(* Visualisation AMAININTERFACE
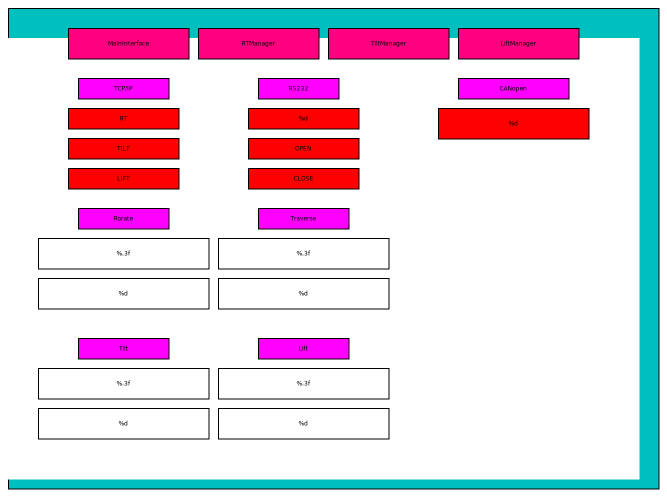
rounded rectangle at (60,20)-(181,51): text "MainInterface"; opens aMainInterface
rounded rectangle at (190,20)-(311,51): text "RTManager"; opens bRTManager
rounded rectangle at (320,20)-(441,51): text "TiltManager"; opens TiltManager
rounded rectangle at (450,20)-(571,51): text "LiftManager"; opens LiftManager
rounded rectangle at (450,70)-(561,91): text "CANopen"
rounded rectangle at (250,70)-(331,91): text "RS232"
rounded rectangle at (70,70)-(161,91): text "TCP/IP"
rounded rectangle at (70,200)-(161,221): text "Rorate"
rounded rectangle at (250,200)-(341,221): text "Traverse"
rounded rectangle at (70,330)-(161,351): text "Tilt"
rounded rectangle at (250,330)-(341,351): text "Lift"
rounded rectangle at (30,360)-(201,391): text "%.3f"
rounded rectangle at (210,360)-(381,391): text "%.3f"; shows .ENC_POS1/100.0
rounded rectangle at (30,400)-(201,431): text "%d"; shows .diActVelocity1/(-2000)
rounded rectangle at (210,400)-(381,431): text "%d"; shows .diActVelocity2/3360
rounded rectangle at (210,230)-(381,261): text "%.3f"; shows .ENC_POS1/100.0
rounded rectangle at (30,230)-(201,261): text "%.3f"
rounded rectangle at (30,270)-(201,301): text "%d"; shows .diActVelocity1/(-2000)
rounded rectangle at (210,270)-(381,301): text "%d"; shows .diActVelocity2/3360
rectangle at (430,100)-(581,131): text "%d"; shows pCanOpenNode[0].nStatus; alarm colour if pCanOpenNode[0].nStatus=5
rounded rectangle at (240,100)-(351,121): text "%d"; shows ComHandle; alarm colour if ComHandle>0
rounded rectangle at (240,130)-(351,151): text "OPEN"; alarm colour if PLC_PRG.open
rounded rectangle at (240,160)-(351,181): text "CLOSE"; alarm colour if PLC_PRG.close
rounded rectangle at (60,100)-(171,121): text "RT"; alarm colour if Client0.diSocket<>-1
rounded rectangle at (60,130)-(171,151): text "TILT"; alarm colour if Client1.diSocket<>-1
rounded rectangle at (60,160)-(171,181): text "LIFT"; alarm colour if Client2.diSocket<>-1
7 more shapes without text or variables
*)

(* Visualisation bRTManager
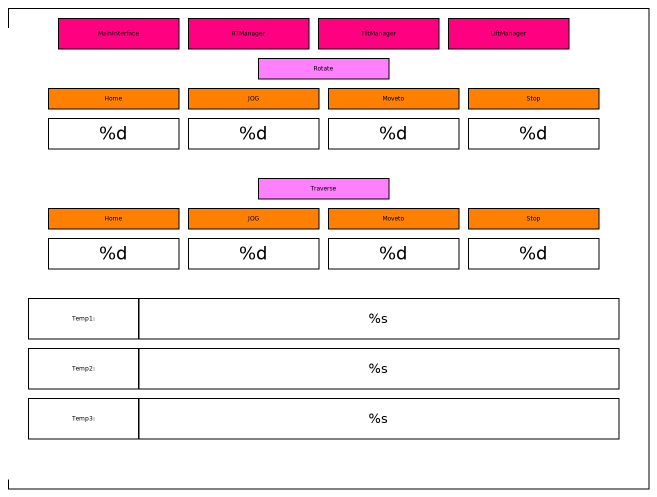
rectangle at (130,340)-(611,381): text "%s"; shows RT_Manager.Temp2
rectangle at (130,390)-(611,431): text "%s"; shows RT_Manager.Temp3
rectangle at (130,290)-(611,331): text "%s"; shows RT_Manager.Temp
rounded rectangle at (250,170)-(381,191): text "Traverse"
rounded rectangle at (40,200)-(171,221): text "Home"
rounded rectangle at (180,200)-(311,221): text "JOG"
rounded rectangle at (320,200)-(451,221): text "Moveto"
rounded rectangle at (460,200)-(591,221): text "Stop"
rectangle at (40,230)-(171,261): text "%d"; shows RT_Manager.diTraverseHomestep
rectangle at (180,230)-(311,261): text "%d"; shows RT_Manager.diTraverseJogstep
rectangle at (320,230)-(451,261): text "%d"; shows RT_Manager.diTraverseMovetostep
rectangle at (460,230)-(591,261): text "%d"; shows RT_Manager.diTraverseStopstep
rectangle at (20,290)-(131,331): text "Temp1:"
rectangle at (20,340)-(131,381): text "Temp2:"
rectangle at (20,390)-(131,431): text "Temp3:"
rounded rectangle at (250,50)-(381,71): text "Rotate"
rounded rectangle at (40,80)-(171,101): text "Home"
rounded rectangle at (180,80)-(311,101): text "JOG"
rounded rectangle at (320,80)-(451,101): text "Moveto"
rounded rectangle at (460,80)-(591,101): text "Stop"
rectangle at (40,110)-(171,141): text "%d"; shows RT_Manager.diRotateHomestep
rectangle at (180,110)-(311,141): text "%d"; shows RT_Manager.diRotateJogstep
rectangle at (320,110)-(451,141): text "%d"; shows RT_Manager.diRotateMovetostep
rectangle at (460,110)-(591,141): text "%d"; shows RT_Manager.diRotateStopstep
rounded rectangle at (180,10)-(301,41): text "RTManager"; opens bRTManager
rounded rectangle at (310,10)-(431,41): text "TiltManager"; opens TiltManager
rounded rectangle at (440,10)-(561,41): text "LiftManager"; opens LiftManager
rounded rectangle at (50,10)-(171,41): text "MainInterface"; opens aMainInterface
4 more shapes without text or variables
*)

(* Visualisation LiftManager
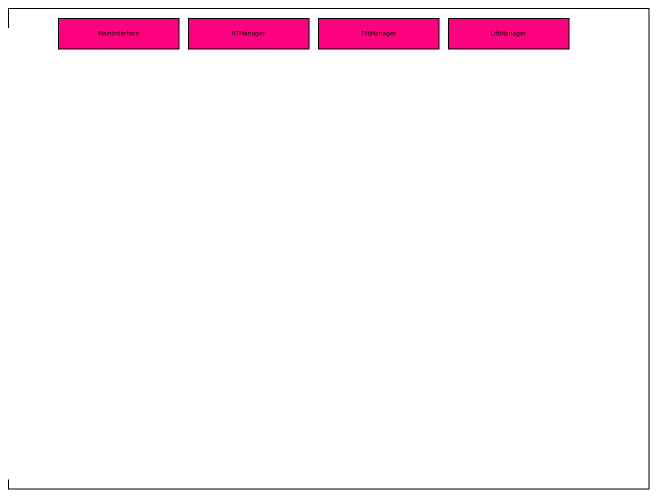
rounded rectangle at (180,10)-(301,41): text "RTManager"; opens bRTManager
rounded rectangle at (310,10)-(431,41): text "TiltManager"; opens TiltManager
rounded rectangle at (440,10)-(561,41): text "LiftManager"; opens LiftManager
rounded rectangle at (50,10)-(171,41): text "MainInterface"; opens aMainInterface
2 more shapes without text or variables
*)

(* Visualisation TiltManager
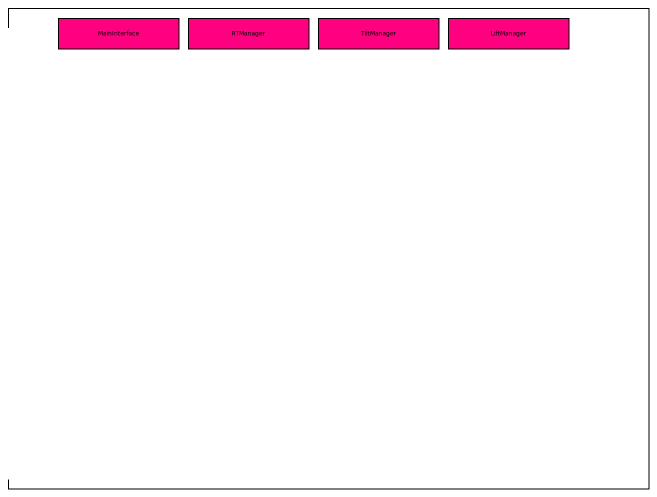
rounded rectangle at (180,10)-(301,41): text "RTManager"; opens bRTManager
rounded rectangle at (310,10)-(431,41): text "TiltManager"; opens TiltManager
rounded rectangle at (440,10)-(561,41): text "LiftManager"; opens LiftManager
rounded rectangle at (50,10)-(171,41): text "MainInterface"; opens aMainInterface
2 more shapes without text or variables
*)
